DATA_BLOCK "ST10_DBInterface_Stopper"
VAR
  Stopper : Array[1..50] of "UDT_StopperInterface";
END_VAR
BEGIN
END_DATA_BLOCK
